// TIA Portal V16 export
// export: Created 2022-02-04T14:40:08.991146Z, ExportSetting WithDefaults, DisplayName Totally Integrated Automation Portal, DisplayVersion V16 Update 1, DisplayName TIA Portal Version Control Interface, DisplayVersion V16, DisplayName TIA Portal Openness, DisplayVersion V16, DisplayName SINAMICS Startdrive Advanced, DisplayVersion V16 Update 5, DisplayName SINAMICS Startdrive G130, G150, S120, S150, SINAMICS MV, S210, DisplayVersion V16 Update 5, DisplayName SINAMICS Startdrive G110M, G120, G120C, G120D, G120P, G115D, DisplayVersion V16 Update 5, DisplayName STEP 7 Professional, DisplayVersion V16, DisplayName STEP 7 Safety, DisplayVersion V16, DisplayName WinCC Advanced, DisplayVersion V16, DisplayName SIMATIC Visualization Architect, DisplayVersion V16
ORGANIZATION_BLOCK "BREAKUP ERROR"   // OB88, LAD, ProcessingInterrupt
TITLE = "Breakup Error"
VERSION : 0.1
// stored: IsIECCheckEnabled false
   VAR_TEMP
      OB88_EV_CLASS : Byte;   // 16#35 Event class 2, Entering event state, Internal fault event
      OB88_SW_FLT : Byte;   // 16#XX, Software programming fault
      OB88_PRIORITY : Byte;   // Priority of OB Execution
      OB88_OB_NUMBR : Byte;   // 88 (Organization block 88, OB88)
      OB88_BLK_TYPE : Byte;   // 16#88/8C/8E Type of block where breakup occured
      OB88_RESERVED_1 : Byte;   // Reserved for system
      OB88_FLT_PRIORITY : Byte;   // Priority of OB caused breakup
      OB88_FLT_OB_NUMBR : Byte;   // OB execution caused breakup
      OB88_BLK_NUM : Word;   // Number of block where breakup occured
      OB88_PRG_ADDR : Word;   // Address in block where breakup occured
      OB88_DATE_TIME : Date_And_Time;   // Date and time OB88 started
   END_VAR
BEGIN
END_ORGANIZATION_BLOCK
